(* IEC 61131-3 sources: JaccoSigma/tempclass/Class/MyObject, 1 file *)

(* ---- MyObject.st ---- *)
(*!
<Class
	Name               = "MyObject"
	Revision           = "0.0"
	RealtimeTask       = "false"
	CyclicTask         = "false"
	BackgroundTask     = "false"
	Sigmatek           = "false"
	OSInterface        = "false"
	HighPriority       = "false"
	Automatic          = "false"
	UpdateMode         = "Prescan"
	SharedCommandTable = "true"
	Objectsize         = "(284,120)">
	<Channels>
		<Server Name="ClassSvr" Visualized="false" Initialize="false" WriteProtected="true" Retentive="false"/>
	</Channels>
</Class>
*)
MyObject : CLASS
  //Servers:
	ClassSvr 	: SvrChCmd_DINT;
  //Clients:
  //Variables:
  //Functions:

	FUNCTION VIRTUAL GLOBAL AddValue
		VAR_INPUT
			Value 	: DINT;
		END_VAR
		VAR_OUTPUT
			Result 	: DINT;
		END_VAR;
  //Tables:
	FUNCTION @STD
		VAR_OUTPUT
			ret_code	: CONFSTATES;
		END_VAR;
	FUNCTION GLOBAL TAB @CT_;
END_CLASS;

FUNCTION VIRTUAL GLOBAL MyObject::AddValue
	VAR_INPUT
		Value 	: DINT;
	END_VAR
	VAR_OUTPUT
		Result 	: DINT;
	END_VAR

  ClassSvr  += Value;
  Result    := ClassSvr;

END_FUNCTION
